FUNCTION A_SINT : ST_Arg
VAR_INPUT
	nNumber	: REFERENCE TO SINT;
END_VAR

IF __ISVALIDREF(nNumber) THEN
	A_SINT.eType := E_ArgType.SIntArg;
	A_SINT.pData := ADR(nNumber);
	A_SINT.nSize := SIZEOF(SINT);
END_IF

END_FUNCTION

(* stored: Version 1.1.0.1, ProductVersion 3.1.4024.15
   POU A_SINT: Id {992a1ab8-5133-424e-abd5-4e1744f29342}, SpecialFunc None *)
